(* global variable list RobotLibraryParameter *)
{attribute 'qualified_only'}
// ------------------------------------------------------------------------- 
//  SRCI Robot Library                                                
// ------------------------------------------------------------------------- 
//                                                                           
//  Object:      Parameter                                       
//  Author:      Thorsten Brach                                                
//  Date:        2024-06-01
//
//  Description:                                              
//   
//                                                                           
//  Copyright: 
//    (C) 2024 Thorsten Brach. All rights reserved                                                                                                                                            
//             Licensed under the MIT License.
//                                                                           
//  Disclaimer:                                                                           
//    This project is provided without any guarantee and can be used for   
//    private and commercial purposes. Any use is at the user’s 
//    own risk and responsibility.
//
// -------------------------------------------------------------------------
VAR_GLOBAL CONSTANT
  /// Maximal amount of tools
  TOOL_MAX                            : DINT := 16;
  /// Maximal amount of frames
  FRAME_MAX                           : DINT := 16;
  /// Maximal amount of loads
  LOAD_MAX                            : DINT := 16;  
  /// Maximal amount of work areas
  WORK_AREAS_MAX                      : DINT := 16;  
  /// Maximal amount of system logs
  SYSTEM_LOG_MAX                      : DINT := 32;  
  /// Maximal amount of message logs
  MESSAGE_LOG_MAX                     : DINT := 100;  
  /// Maximum string length for message texts
  MESSAGE_TEXT_LEN                    : DINT := 255;
  /// Maximal amount of List entries 
  LIST_ENTRIES_MAX                    : DINT := 100;
  /// Maximal amount of bytes for the parameter payload
  PARAMETER_PAYLOAD_MAX               : DINT := 255;  
  /// Maximal amount of bytes for the response payload
  RESPONSE_PAYLOAD_MAX                : DINT := 255;  
  /// Maximal amount of bytes that can be exchanged with the sub program on the RC
  SUB_PROGRAM_DATA_MAX                : DINT := 189;
  /// Maximal amount of spline data
  SPLINE_DATA_MAX                     : DINT := 64;
  /// Maximal amount of entries in the Active Command Register
  ACTIVE_CMD_REGISTER_ENTRIES_MAX     : DINT := 50;
  /// Maximal amount of message codes
  MESSAGE_CODES_MAX                   : DINT := 15;
  /// Maximal amount of fragments
  FRAGMENT_MAX                        : DINT := 9;
  /// Flag to indicate that the byte order must be changed
  SWAP_BYTE_ORDER                     : BOOL := TRUE; 
  /// Timeout for checking for invalid frames
  INVALID_FRAMES_CHECK_TIMEOUT        : TIME := T#60S;
  /// Warning limit for ACR registers running low
  ACR_USAGE_WARNING_LIMIT             : REAL := 80.0;  
END_VAR

INTERFACE IMessageLogger
METHOD PUBLIC AddMessageLog
VAR_INPUT
  /// Message to add to the log
  MessageLog : AlarmMessage;
END_VAR
END_METHOD
METHOD PUBLIC AddSystemLog
VAR_INPUT
  /// System messafe to add to the log
  SystemLog : STRING(RobotLibraryParameter.MESSAGE_TEXT_LEN);
END_VAR
END_METHOD
END_INTERFACE

INTERFACE IRobotLibraryCommandFB
METHOD PUBLIC CallBack : DINT
VAR_INPUT
  /// Response data
  RspData : AxesGroupAcyclicAcrEntryRspBuffer;  
END_VAR
END_METHOD
PROPERTY CommandData : RobotLibrarySendDataFB
END_PROPERTY
END_INTERFACE

FUNCTION IsDefaultDynamicsEqual : BOOL
// ------------------------------------------------------------------------- 
//  SRCI Robot Library                                                
// ------------------------------------------------------------------------- 
//                                                                           
//  Object:      IsDefaultDynamicsEqual                                       
//  Author:      Thorsten Brach                                                
//  Date:        2025-04-23
//
//  Description:                                              
//   
//                                                                           
//  Copyright: 
//    (C) 2025 Thorsten Brach. All rights reserved                                                                                                                                            
//             Licensed under the MIT License.
//                                                                           
//  Disclaimer:                                                                           
//    This project is provided without any guarantee and can be used for   
//    private and commercial purposes. Any use is at the user’s 
//    own risk and responsibility.
//
// -------------------------------------------------------------------------
VAR_INPUT
  /// DefaultDynamics 1 to compare
  Data1           : DefaultDynamics;
  /// DefaultDynamics 2 to compare
  Data2           : DefaultDynamics;
  /// Flag to ignore the timestamp during the comparison
  IgnoreTimestamp : BOOL;
END_VAR

            IF (IgnoreTimestamp)
THEN
  Data1.Timestamp := Data2.Timestamp;
END_IF                    
                    
IsDefaultDynamicsEqual := ( SysDepMemCmp( pData1 := ADR(Data1), pData2 :=  ADR(Data2), DataLen := SIZEOF(Data1)) = RobotLibraryConstants.OK );
          
END_FUNCTION

FUNCTION IsFrameDataEqual : BOOL
// ------------------------------------------------------------------------- 
//  SRCI Robot Library                                                
// ------------------------------------------------------------------------- 
//                                                                           
//  Object:      IsFrameDataEqual                                       
//  Author:      Thorsten Brach                                                
//  Date:        2025-04-23
//
//  Description:                                              
//   
//                                                                           
//  Copyright: 
//    (C) 2025 Thorsten Brach. All rights reserved                                                                                                                                            
//             Licensed under the MIT License.
//                                                                           
//  Disclaimer:                                                                           
//    This project is provided without any guarantee and can be used for   
//    private and commercial purposes. Any use is at the user’s 
//    own risk and responsibility.
//
// -------------------------------------------------------------------------
VAR_INPUT
  /// FrameData 1 to compare
  Data1           : FrameData;
  /// FrameData 2 to compare
  Data2           : FrameData;
  /// Flag to ignore the timestamp during the comparison
  IgnoreTimestamp : BOOL;
END_VAR

            IF (IgnoreTimestamp)
THEN
  Data1.Timestamp := Data2.Timestamp;
END_IF                    
                    
IsFrameDataEqual := ( SysDepMemCmp( pData1 := ADR(Data1), pData2 :=  ADR(Data2), DataLen := SIZEOF(Data1)) = RobotLibraryConstants.OK );                    
          
END_FUNCTION

FUNCTION IsLoadDataEqual : BOOL
// ------------------------------------------------------------------------- 
//  SRCI Robot Library                                                
// ------------------------------------------------------------------------- 
//                                                                           
//  Object:      IsLoadDataEqual                                       
//  Author:      Thorsten Brach                                                
//  Date:        2025-04-23
//
//  Description:                                              
//   
//                                                                           
//  Copyright: 
//    (C) 2025 Thorsten Brach. All rights reserved                                                                                                                                            
//             Licensed under the MIT License.
//                                                                           
//  Disclaimer:                                                                           
//    This project is provided without any guarantee and can be used for   
//    private and commercial purposes. Any use is at the user’s 
//    own risk and responsibility.
//
// -------------------------------------------------------------------------
VAR_INPUT
  /// LoadData 1 to compare
  Data1           : LoadData;
  /// LoadData 2 to compare
  Data2           : LoadData;
  /// Flag to ignore the timestamp during the comparison
  IgnoreTimestamp : BOOL;
END_VAR

            IF (IgnoreTimestamp)
THEN
  Data1.Timestamp := Data2.Timestamp;
END_IF                    
                    
IsLoadDataEqual := ( SysDepMemCmp( pData1 := ADR(Data1), pData2 :=  ADR(Data2), DataLen := SIZEOF(Data1)) = RobotLibraryConstants.OK );
          
END_FUNCTION

FUNCTION IsReferenceDynamicsEqual : BOOL
// ------------------------------------------------------------------------- 
//  SRCI Robot Library                                                
// ------------------------------------------------------------------------- 
//                                                                           
//  Object:      IsReferenceDynamicsEqual                                       
//  Author:      Thorsten Brach                                                
//  Date:        2025-04-23
//
//  Description:                                              
//   
//                                                                           
//  Copyright: 
//    (C) 2025 Thorsten Brach. All rights reserved                                                                                                                                            
//             Licensed under the MIT License.
//                                                                           
//  Disclaimer:                                                                           
//    This project is provided without any guarantee and can be used for   
//    private and commercial purposes. Any use is at the user’s 
//    own risk and responsibility.
//
// -------------------------------------------------------------------------
VAR_INPUT
  /// ReferenceDynamics 1 to compare
  Data1           : ReferenceDynamics;
  /// ReferenceDynamics 2 to compare
  Data2           : ReferenceDynamics;
  /// Flag to ignore the timestamp during the comparison
  IgnoreTimestamp : BOOL;
END_VAR

            IF (IgnoreTimestamp)
THEN
  Data1.Timestamp := Data2.Timestamp;
END_IF                    
                    
IsReferenceDynamicsEqual := ( SysDepMemCmp( pData1 := ADR(Data1), pData2 :=  ADR(Data2), DataLen := SIZEOF(Data1)) = RobotLibraryConstants.OK );
          
END_FUNCTION

FUNCTION IsSwLimitsEqual : BOOL
// ------------------------------------------------------------------------- 
//  SRCI Robot Library                                                
// ------------------------------------------------------------------------- 
//                                                                           
//  Object:      IsSwLimitsEqual                                       
//  Author:      Thorsten Brach                                                
//  Date:        2025-04-23
//
//  Description:                                              
//   
//                                                                           
//  Copyright: 
//    (C) 2025 Thorsten Brach. All rights reserved                                                                                                                                            
//             Licensed under the MIT License.
//                                                                           
//  Disclaimer:                                                                           
//    This project is provided without any guarantee and can be used for   
//    private and commercial purposes. Any use is at the user’s 
//    own risk and responsibility.
//
// -------------------------------------------------------------------------
VAR_INPUT
  /// SW Limit 1 to compare
  Data1           : SWLimits;
  /// SW LIMIT 2 to compare
  Data2           : SWLimits;
  /// Flag to ignore the timestamp during the comparison
  IgnoreTimestamp : BOOL;
END_VAR

            IF (IgnoreTimestamp)
THEN
  Data1.Timestamp := Data2.Timestamp;
END_IF                    
                    
IsSwLimitsEqual := ( SysDepMemCmp( pData1 := ADR(Data1), pData2 :=  ADR(Data2), DataLen := SIZEOF(Data1)) = RobotLibraryConstants.OK );
          
END_FUNCTION

FUNCTION IsToolDataEqual : BOOL
// ------------------------------------------------------------------------- 
//  SRCI Robot Library                                                
// ------------------------------------------------------------------------- 
//                                                                           
//  Object:      IsToolDataEqual                                       
//  Author:      Thorsten Brach                                                
//  Date:        2025-04-23
//
//  Description:                                              
//   
//                                                                           
//  Copyright: 
//    (C) 2025 Thorsten Brach. All rights reserved                                                                                                                                            
//             Licensed under the MIT License.
//                                                                           
//  Disclaimer:                                                                           
//    This project is provided without any guarantee and can be used for   
//    private and commercial purposes. Any use is at the user’s 
//    own risk and responsibility.
//
// -------------------------------------------------------------------------
VAR_INPUT
  /// ToolData 1 to compare
  Data1           : ToolData;
  /// ToolData 2 to compare
  Data2           : ToolData;
  /// Flag to ignore the timestamp during the comparison
  IgnoreTimestamp : BOOL;
END_VAR

            IF (IgnoreTimestamp)
THEN
  Data1.Timestamp := Data2.Timestamp;
END_IF                    
                    
IsToolDataEqual := ( SysDepMemCmp( pData1 := ADR(Data1), pData2 :=  ADR(Data2), DataLen := SIZEOF(Data1)) = RobotLibraryConstants.OK );                    
          
END_FUNCTION

FUNCTION IsWorkAreaEqual : BOOL
// ------------------------------------------------------------------------- 
//  SRCI Robot Library                                                
// ------------------------------------------------------------------------- 
//                                                                           
//  Object:      IsWorkAreaEqual                                       
//  Author:      Thorsten Brach                                                
//  Date:        2025-04-23
//
//  Description:                                              
//   
//                                                                           
//  Copyright: 
//    (C) 2025 Thorsten Brach. All rights reserved                                                                                                                                            
//             Licensed under the MIT License.
//                                                                           
//  Disclaimer:                                                                           
//    This project is provided without any guarantee and can be used for   
//    private and commercial purposes. Any use is at the user’s 
//    own risk and responsibility.
//
// -------------------------------------------------------------------------
VAR_INPUT
  /// WorkArea 1 to compare
  Data1           : RobotWorkAreaData;
  /// WorkArea 2 to compare
  Data2           : RobotWorkAreaData;
  /// Flag to ignore the timestamp during the comparison
  IgnoreTimestamp : BOOL;
END_VAR

            IF (IgnoreTimestamp)
THEN
  Data1.Timestamp := Data2.Timestamp;
END_IF                    
                    
IsWorkAreaEqual := ( SysDepMemCmp( pData1 := ADR(Data1), pData2 :=  ADR(Data2), DataLen := SIZEOF(Data1)) = RobotLibraryConstants.OK );
          
END_FUNCTION

FUNCTION CheckTimeout : DINT
// ------------------------------------------------------------------------- 
//  SRCI Robot Library                                                
// ------------------------------------------------------------------------- 
//                                                                           
//  Object:      SwapBytes                                       
//  Author:      Thorsten Brach                                                
//  Date:        2024-12-18
//
//  Description:                                              
//   
//                                                                           
//  Copyright: 
//    (C) 2024 Thorsten Brach. All rights reserved                                                                                                                                            
//             Licensed under the MIT License.
//                                                                           
//  Disclaimer:                                                                           
//    This project is provided without any guarantee and can be used for   
//    private and commercial purposes. Any use is at the user’s 
//    own risk and responsibility.
//
// -------------------------------------------------------------------------
VAR_INPUT
  /// Reference to TON instance
  rTimer : REFERENCE TO TON;
END_VAR

            // Call timer 
rTimer();

// check if timer elapsed
IF (rTimer.Q = TRUE)
THEN
  // assign return value
  CheckTimeout := RobotLibraryConstants.OK;
ELSE
  // assign return value
  CheckTimeout := RobotLibraryConstants.RUNNING;
END_IF
          
END_FUNCTION

FUNCTION SetTimeout : DINT
// ------------------------------------------------------------------------- 
//  SRCI Robot Library                                                
// ------------------------------------------------------------------------- 
//                                                                           
//  Object:      SwapBytes                                       
//  Author:      Thorsten Brach                                                
//  Date:        2024-12-18
//
//  Description:                                              
//   
//                                                                           
//  Copyright: 
//    (C) 2024 Thorsten Brach. All rights reserved                                                                                                                                            
//             Licensed under the MIT License.
//                                                                           
//  Disclaimer:                                                                           
//    This project is provided without any guarantee and can be used for   
//    private and commercial purposes. Any use is at the user’s 
//    own risk and responsibility.
//
// -------------------------------------------------------------------------
VAR_INPUT
  /// Timeout to be set
  PT     : TIME;
  /// Reference to TON instance
  rTimer : REFERENCE TO TON;
END_VAR

            rTimer(IN := FALSE);          // Reset timer
rTimer(PT := PT, IN := TRUE); // Start timer

// assign return value
SetTimeout := RobotLibraryConstants.OK;
          
END_FUNCTION

FUNCTION DATE_TO_IEC_DATE : IEC_DATE
// ------------------------------------------------------------------------- 
//  SRCI Robot Library                                                
// ------------------------------------------------------------------------- 
//                                                                           
//  Object:      DATE_TO_IEC_DATE                                       
//  Author:      Thorsten Brach                                                
//  Date:        2024-06-01
//
//  Description:                                              
//   
//                                                                           
//  Copyright: 
//    (C) 2024 Thorsten Brach. All rights reserved                                                                                                                                            
//             Licensed under the MIT License.
//                                                                           
//  Disclaimer:                                                                           
//    This project is provided without any guarantee and can be used for   
//    private and commercial purposes. Any use is at the user’s 
//    own risk and responsibility.
//
// -------------------------------------------------------------------------
VAR_INPUT
  Value    : DATE;
END_VAR

VAR
 _tmpDate1 : DWORD;
 _tmpDate2 : DWORD;
 _initDate : DATE := DATE#1990-01-01;
 END_VAR

            // Siemens Dateformat is Day since 01.01.1990
// TwinCat Dateformat is seconds sinde 01.01.1970
// Calculation : 
// ( [TwinCat current date] - [ TwinCat 01.01.1970] ) / [Seconds a Day] = Days sinde 01.01.1990 (Siemens Format)

// copy date to dword
SysDepMemCpy( pDest := ADR(_tmpDate1), pSrc := ADR( Value   ), DataLen := SIZEOF( Value   ));
// copy date to dword
SysDepMemCpy( pDest := ADR(_tmpDate2), pSrc := ADR(_initDate), DataLen := SIZEOF(_initDate));

// calculate IEC Date :  
DATE_TO_IEC_DATE := UDINT_TO_UINT((_tmpDate1 - _tmpDate2) / 86400); // 86400 Seconds = 1 day 

          
END_FUNCTION

FUNCTION IEC_DATE_TO_DATE : DATE
// ------------------------------------------------------------------------- 
//  SRCI Robot Library                                                
// ------------------------------------------------------------------------- 
//                                                                           
//  Object:      IEC_DATE_TO_DATE                                       
//  Author:      Thorsten Brach                                                
//  Date:        2025-01-05
//
//  Description:                                              
//   
//                                                                           
//  Copyright: 
//    (C) 2025 Thorsten Brach. All rights reserved                                                                                                                                            
//             Licensed under the MIT License.
//                                                                           
//  Disclaimer:                                                                           
//    This project is provided without any guarantee and can be used for   
//    private and commercial purposes. Any use is at the user’s 
//    own risk and responsibility.
//
// -------------------------------------------------------------------------
VAR_INPUT
  Value    : IEC_DATE;
END_VAR

VAR
 _tmpDate1 : DWORD;
 _initDate : DATE := DATE#1990-01-01;
 END_VAR

            // Siemens Dateformat is Day since 01.01.1990
// TwinCat Dateformat is seconds sinde 01.01.1970
// Calculation : 
// ( [ TwinCat 01.01.1990] + [IEC Date]) * [Seconds a Day] = (TwinCat Format)

// copy date to dword
SysDepMemCpy( pDest := ADR(_tmpDate1), pSrc := ADR( _initDate ), DataLen := SIZEOF( _initDate ));

// calculate IEC Date :  
IEC_DATE_TO_DATE := DWORD_TO_DATE( _tmpDate1 + ( Value * 86400)); // 86400 Seconds = 1 day 
          
END_FUNCTION

FUNCTION IEC_TIME_TO_TIME : TOD
// ------------------------------------------------------------------------- 
//  SRCI Robot Library                                                
// ------------------------------------------------------------------------- 
//                                                                           
//  Object:      IEC_TIME_TO_TIME                                       
//  Author:      Thorsten Brach                                                
//  Date:        2025-01-05
//
//  Description:                                              
//   
//                                                                           
//  Copyright: 
//    (C) 2025 Thorsten Brach. All rights reserved                                                                                                                                            
//             Licensed under the MIT License.
//                                                                           
//  Disclaimer:                                                                           
//    This project is provided without any guarantee and can be used for   
//    private and commercial purposes. Any use is at the user’s 
//    own risk and responsibility.
//
// -------------------------------------------------------------------------
VAR_INPUT
  Value : IEC_TIME;
END_VAR

            IEC_TIME_TO_TIME := Value; 
          
END_FUNCTION

FUNCTION IEC_TIMESTAMP_TO_DT : DT
// ------------------------------------------------------------------------- 
//  SRCI Robot Library                                                
// ------------------------------------------------------------------------- 
//                                                                           
//  Object:      TIME_TO_IEC_TIME                                       
//  Author:      Thorsten Brach                                                
//  Date:        2025-01-05
//
//  Description:                                              
//   
//                                                                           
//  Copyright: 
//    (C) 2025 Thorsten Brach. All rights reserved                                                                                                                                            
//             Licensed under the MIT License.
//                                                                           
//  Disclaimer:                                                                           
//    This project is provided without any guarantee and can be used for   
//    private and commercial purposes. Any use is at the user’s 
//    own risk and responsibility.
//
// -------------------------------------------------------------------------
VAR_INPUT
  Value : IEC_TIMESTAMP;
END_VAR

VAR
  /// internal date
 _date    : DATE;
  /// internal date as string
 _dateStr : STRING;
  /// internal time
 _time    : TOD;
  /// internal time as string
 _timeStr : STRING;
END_VAR

            _date := IEC_DATE_TO_DATE(Value.IEC_DATE); 
_time := IEC_TIME_TO_TIME(Value.IEC_TIME); 


// Example : DATE#2025-1-5
_dateStr := DATE_TO_STRING(_date);
// Example : DT#2025-1-5
_dateStr := strReplace(_dateStr, 'D#', 'DT#');

// Example : TOD#15:18:4.567
_timeStr :=  TOD_TO_STRING(_time);
// Example : -15:18:4.567
_timeStr := strReplace(_timeStr, 'TOD#', '-');

// Example : DT#2025-1-5-15:18:4.567
IEC_TIMESTAMP_TO_DT := STRING_TO_DT( Concat(_dateStr,_timeStr));
          
END_FUNCTION

FUNCTION IEC_TIMESTAMP_TO_SYSTEMTIME : SystemTime
// ------------------------------------------------------------------------- 
//  SRCI Robot Library                                                
// ------------------------------------------------------------------------- 
//                                                                           
//  Object:      IEC_TIMESTAMP_TO_SYSTEMTIME                                       
//  Author:      Thorsten Brach                                                
//  Date:        2025-01-05
//
//  Description:                                              
//   
//                                                                           
//  Copyright: 
//    (C) 2025 Thorsten Brach. All rights reserved                                                                                                                                            
//             Licensed under the MIT License.
//                                                                           
//  Disclaimer:                                                                           
//    This project is provided without any guarantee and can be used for   
//    private and commercial purposes. Any use is at the user’s 
//    own risk and responsibility.
//
// -------------------------------------------------------------------------
VAR_INPUT
  Value : IEC_TIMESTAMP;
END_VAR

VAR
  /// internal date
 _date    : DATE;
  /// internal date as string
 _dateStr : STRING;
  /// internal time
 _time    : TOD;
  /// internal time as string
 _timeStr : STRING;
END_VAR

            IEC_TIMESTAMP_TO_SYSTEMTIME.SystemDate := IEC_DATE_TO_DATE(Value.IEC_DATE);
IEC_TIMESTAMP_TO_SYSTEMTIME.SystemTime := IEC_TIME_TO_TIME(Value.IEC_TIME);
          
END_FUNCTION

FUNCTION SYSTEMTIME_TO_IEC_TIMESTAMP : IEC_TIMESTAMP
// ------------------------------------------------------------------------- 
//  SRCI Robot Library                                                
// ------------------------------------------------------------------------- 
//                                                                           
//  Object:      SYSTEMTIME_TO_IEC_TIMESTAMP                                       
//  Author:      Thorsten Brach                                                
//  Date:        2025-03-30
//
//  Description:                                              
//   
//                                                                           
//  Copyright: 
//    (C) 2025 Thorsten Brach. All rights reserved                                                                                                                                            
//             Licensed under the MIT License.
//                                                                           
//  Disclaimer:                                                                           
//    This project is provided without any guarantee and can be used for   
//    private and commercial purposes. Any use is at the user’s 
//    own risk and responsibility.
//
// -------------------------------------------------------------------------
VAR_INPUT
  SystemTime : SystemTime;
END_VAR

            SYSTEMTIME_TO_IEC_TIMESTAMP.IEC_DATE := DATE_TO_IEC_DATE(SystemTime.SystemDate);
SYSTEMTIME_TO_IEC_TIMESTAMP.IEC_TIME := TIME_TO_IEC_TIME(SystemTime.SystemTime);

          
END_FUNCTION

FUNCTION TIME_TO_IEC_TIME : IEC_TIME
// ------------------------------------------------------------------------- 
//  SRCI Robot Library                                                
// ------------------------------------------------------------------------- 
//                                                                           
//  Object:      TIME_TO_IEC_TIME                                       
//  Author:      Thorsten Brach                                                
//  Date:        2024-06-01
//
//  Description:                                              
//   
//                                                                           
//  Copyright: 
//    (C) 2024 Thorsten Brach. All rights reserved                                                                                                                                            
//             Licensed under the MIT License.
//                                                                           
//  Disclaimer:                                                                           
//    This project is provided without any guarantee and can be used for   
//    private and commercial purposes. Any use is at the user’s 
//    own risk and responsibility.
//
// -------------------------------------------------------------------------
VAR_INPUT
  Value : TOD;
END_VAR

            TIME_TO_IEC_TIME := Value; 
          
END_FUNCTION

FUNCTION ArmConfigParameterToBytes : ARRAY[0..1] of BYTE
// ------------------------------------------------------------------------- 
//  SRCI Robot Library                                                
// ------------------------------------------------------------------------- 
//                                                                           
//  Object:      ArmConfigParameterToBytes                                       
//  Author:      Thorsten Brach                                                
//  Date:        2025-01-30
//
//  Description:                                              
//   
//                                                                           
//  Copyright: 
//    (C) 2025 Thorsten Brach. All rights reserved                                                                                                                                            
//             Licensed under the MIT License.
//                                                                           
//  Disclaimer:                                                                           
//    This project is provided without any guarantee and can be used for   
//    private and commercial purposes. Any use is at the user’s 
//    own risk and responsibility.
//
// -------------------------------------------------------------------------
VAR_INPUT
 /// ArmConfigParameter
 Value: ArmConfigParameter;
END_VAR

            ArmConfigParameterToBytes[0].0 := Value.Shoulder.0;
ArmConfigParameterToBytes[0].1 := Value.Shoulder.1;
ArmConfigParameterToBytes[0].2 := Value.Shoulder.2;
ArmConfigParameterToBytes[0].3 := Value.Shoulder.3;
ArmConfigParameterToBytes[0].4 := Value.Elbow.0;
ArmConfigParameterToBytes[0].5 := Value.Elbow.1;
ArmConfigParameterToBytes[0].6 := Value.Elbow.2;
ArmConfigParameterToBytes[0].7 := Value.Elbow.3;
ArmConfigParameterToBytes[1].0 := Value.Wrist.0;
ArmConfigParameterToBytes[1].1 := Value.Wrist.1;
ArmConfigParameterToBytes[1].2 := Value.Wrist.2;
ArmConfigParameterToBytes[1].3 := Value.Wrist.3;
ArmConfigParameterToBytes[1].4 := FALSE;
ArmConfigParameterToBytes[1].5 := FALSE;
ArmConfigParameterToBytes[1].6 := FALSE;
ArmConfigParameterToBytes[1].7 := FALSE;
          
END_FUNCTION

FUNCTION BytesToRCSupportedFunctions : RCSupportedFunctions
// ------------------------------------------------------------------------- 
//  SRCI Robot Library                                                
// ------------------------------------------------------------------------- 
//                                                                           
//  Object:      BytesToRCSupportedFunctions                                       
//  Author:      Thorsten Brach                                                
//  Date:        2024-12-18
//
//  Description:                                              
//   
//                                                                           
//  Copyright: 
//    (C) 2024 Thorsten Brach. All rights reserved                                                                                                                                            
//             Licensed under the MIT License.
//                                                                           
//  Disclaimer:                                                                           
//    This project is provided without any guarantee and can be used for   
//    private and commercial purposes. Any use is at the user’s 
//    own risk and responsibility.
//
// -------------------------------------------------------------------------
VAR_INPUT
  Bytes : ARRAY [0..18] OF BYTE;
END_VAR

            // Byte 00 - Bit 0  
BytesToRCSupportedFunctions.Reserved                   := Bytes[00].0;
// Byte 00 - Bit 1 
BytesToRCSupportedFunctions.ReadRobotData              := Bytes[00].1;
// Byte 00 - Bit 2  
BytesToRCSupportedFunctions.EnableRobot                := Bytes[00].2;
// Byte 00 - Bit 3  
BytesToRCSupportedFunctions.GroupReset                 := Bytes[00].3;
// Byte 00 - Bit 4  
BytesToRCSupportedFunctions.ReadActualPosition         := Bytes[00].4;
// Byte 00 - Bit 5 
BytesToRCSupportedFunctions.ReadActualPositionCyclic   := Bytes[00].5;
// Byte 00 - Bit 6  
BytesToRCSupportedFunctions.ExchangeConfiguration      := Bytes[00].6;
// Byte 00 - Bit 7  
BytesToRCSupportedFunctions.SetSequence                := Bytes[00].7;

// Byte 01 - Bit 0  
BytesToRCSupportedFunctions.ChangeSpeedOverride        := Bytes[01].0;
// Byte 01 - Bit 1  
BytesToRCSupportedFunctions.ReadMessages               := Bytes[01].1;
// Byte 01 - Bit 2  
BytesToRCSupportedFunctions.ReadRobotReferenceDynamics := Bytes[01].2;
// Byte 01 - Bit 3  
BytesToRCSupportedFunctions.WriteFrameData             := Bytes[01].3;
// Byte 01 - Bit 4  
BytesToRCSupportedFunctions.WriteToolData              := Bytes[01].4;
// Byte 01 - Bit 5  
BytesToRCSupportedFunctions.WriteLoadData              := Bytes[01].5;
// Byte 01 - Bit 6  
BytesToRCSupportedFunctions.WriteRobotReferenceDynamics:= Bytes[01].6;
// Byte 01 - Bit 7  
BytesToRCSupportedFunctions.WriteRobotDefaultDynamics  := Bytes[01].7;

// Byte 02 - Bit 0  
BytesToRCSupportedFunctions.ReadRobotDefaultDynamics   := Bytes[02].0;
// Byte 02 - Bit 1  
BytesToRCSupportedFunctions.ReadFrameData              := Bytes[02].1;
// Byte 02 - Bit 2  
BytesToRCSupportedFunctions.ReadToolData               := Bytes[02].2;
// Byte 02 - Bit 3  
BytesToRCSupportedFunctions.ReadLoadData               := Bytes[02].3;
// Byte 02 - Bit 4  
BytesToRCSupportedFunctions.ReadRobotSWLimits          := Bytes[02].4;
// Byte 02 - Bit 5  
BytesToRCSupportedFunctions.GroupJog                   := Bytes[02].5;
// Byte 02 - Bit 6  
BytesToRCSupportedFunctions.MoveLinearAbsolute         := Bytes[02].6;
// Byte 02 - Bit 7  
BytesToRCSupportedFunctions.MoveDirectAbsolute         := Bytes[02].7;

// Byte 03 - Bit 0  
BytesToRCSupportedFunctions.MoveAxesAbsolute           := Bytes[03].0;
// Byte 03 - Bit 1  
BytesToRCSupportedFunctions.GroupStop                  := Bytes[03].1;
// Byte 03 - Bit 2
BytesToRCSupportedFunctions.GroupContinue              := Bytes[03].2;
// Byte 03 - Bit 3
BytesToRCSupportedFunctions.GroupInterrupt             := Bytes[03].3;
// Byte 03 - Bit 4
BytesToRCSupportedFunctions.ReturnToPrimary            := Bytes[03].4;
// Byte 03 - Bit 5
BytesToRCSupportedFunctions.MoveLinearAbsoluteJ        := Bytes[03].5;
// Byte 03 - Bit 6
BytesToRCSupportedFunctions.MoveDirectRelative         := Bytes[03].6;
// Byte 03 - Bit 7
BytesToRCSupportedFunctions.MoveAxesRelative           := Bytes[03].7;

// Byte 04 - Bit 0
BytesToRCSupportedFunctions.MoveCircularAbsolute       := Bytes[04].0;
// Byte 04 - Bit 1
BytesToRCSupportedFunctions.MoveCircularRelative       := Bytes[04].1;
// Byte 04 - Bit 2
BytesToRCSupportedFunctions.MoveLinearOffset           := Bytes[04].2;
// Byte 04 - Bit 3
BytesToRCSupportedFunctions.MoveDirectOffset           := Bytes[04].3;
// Byte 04 - Bit 4
BytesToRCSupportedFunctions.WaitTime                   := Bytes[04].4;
// Byte 04 - Bit 5
BytesToRCSupportedFunctions.ReadDigitalInputs          := Bytes[04].5;
// Byte 04 - Bit 6
BytesToRCSupportedFunctions.ReadDigitalOutputs         := Bytes[04].6;
// Byte 04 - Bit 7
BytesToRCSupportedFunctions.WriteDigitalOutputs        := Bytes[04].7;

// Byte 05 - Bit 0
BytesToRCSupportedFunctions.ReadIntegers               := Bytes[05].0;
// Byte 05 - Bit 1
BytesToRCSupportedFunctions.ReadReals                  := Bytes[05].1;
// Byte 05 - Bit 2
BytesToRCSupportedFunctions.WriteIntegers              := Bytes[05].2;
// Byte 05 - Bit 3
BytesToRCSupportedFunctions.WriteReals                 := Bytes[05].3;
// Byte 05 - Bit 4
BytesToRCSupportedFunctions.MoveLinearCam              := Bytes[05].4;
// Byte 05 - Bit 5
BytesToRCSupportedFunctions.MoveDirectCam              := Bytes[05].5;
// Byte 05 - Bit 6
BytesToRCSupportedFunctions.MoveCircularCam            := Bytes[05].6;
// Byte 05 - Bit 7
BytesToRCSupportedFunctions.SetTriggerRegister         := Bytes[05].7;

// Byte 06 - Bit 0
BytesToRCSupportedFunctions.SetTriggerLimit            := Bytes[06].0;
// Byte 06 - Bit 1
BytesToRCSupportedFunctions.SetTriggerUser             := Bytes[06].1;
// Byte 06 - Bit 2
BytesToRCSupportedFunctions.SetTriggerError            := Bytes[06].2;
// Byte 06 - Bit 3
BytesToRCSupportedFunctions.ReactAtTrigger             := Bytes[06].3;
// Byte 06 - Bit 4
BytesToRCSupportedFunctions.WaitForTrigger             := Bytes[06].4;
// Byte 06 - Bit 5
BytesToRCSupportedFunctions.ReadSystemVariable         := Bytes[06].5;
// Byte 06 - Bit 6
BytesToRCSupportedFunctions.WriteSystemVariable        := Bytes[06].6;
// Byte 06 - Bit 7
BytesToRCSupportedFunctions.CalculateForwardKinematic  := Bytes[06].7;

// Byte 07 - Bit 0
BytesToRCSupportedFunctions.CalculateInverseKinematic  := Bytes[07].0;
// Byte 07 - Bit 1
BytesToRCSupportedFunctions.CalculateCartesianPosition := Bytes[07].1;
// Byte 07 - Bit 2
BytesToRCSupportedFunctions.CalculateTool              := Bytes[07].2;
// Byte 07 - Bit 3
BytesToRCSupportedFunctions.CalculateFrame             := Bytes[07].3;
// Byte 07 - Bit 4
BytesToRCSupportedFunctions.ActivateNextCommand        := Bytes[07].4;
// Byte 07 - Bit 5
BytesToRCSupportedFunctions.ShiftPosition              := Bytes[07].5;
// Byte 07 - Bit 6
BytesToRCSupportedFunctions.CallSubprogram             := Bytes[07].6;
// Byte 07 - Bit 7
BytesToRCSupportedFunctions.MoveLinearRelative         := Bytes[07].7;

// Byte 08 - Bit 0
BytesToRCSupportedFunctions.WriteCallSubprogramCyclic  := Bytes[08].0;
// Byte 08 - Bit 1
BytesToRCSupportedFunctions.ReadCallSubprogramCyclic   := Bytes[08].1;
// Byte 08 - Bit 2
BytesToRCSupportedFunctions.StopSubprogram             := Bytes[08].2;
// Byte 08 - Bit 3
BytesToRCSupportedFunctions.ReadDHParameter            := Bytes[08].3;
// Byte 08 - Bit 4
BytesToRCSupportedFunctions.RestartController          := Bytes[08].4;
// Byte 08 - Bit 5
BytesToRCSupportedFunctions.ReadActualTCPVelocity      := Bytes[08].5;
// Byte 08 - Bit 6
BytesToRCSupportedFunctions.UserLogin                  := Bytes[08].6;
// Byte 08 - Bit 7
BytesToRCSupportedFunctions.SwitchLanguage             := Bytes[08].7;

// Byte 09 - Bit 0
BytesToRCSupportedFunctions.WriteRobotSWLimits         := Bytes[09].0;
// Byte 09 - Bit 1
BytesToRCSupportedFunctions.SetOperationMode           := Bytes[09].1;
// Byte 09 - Bit 2
BytesToRCSupportedFunctions.ReadWorkArea               := Bytes[09].2;
// Byte 09 - Bit 3
BytesToRCSupportedFunctions.WriteWorkArea              := Bytes[09].3;
// Byte 09 - Bit 4
BytesToRCSupportedFunctions.ActivateWorkArea           := Bytes[09].4;
// Byte 09 - Bit 5
BytesToRCSupportedFunctions.MonitorWorkArea            := Bytes[09].5;
// Byte 09 - Bit 6
BytesToRCSupportedFunctions.MoveApproachLinear         := Bytes[09].6;
// Byte 09 - Bit 7
BytesToRCSupportedFunctions.MoveDepartLinear           := Bytes[09].7;

// Byte 10 - Bit 0
BytesToRCSupportedFunctions.MoveApproachDirect         := Bytes[10].0;
// Byte 10 - Bit 1
BytesToRCSupportedFunctions.MoveDepartDirect           := Bytes[10].1;
// Byte 10 - Bit 2
BytesToRCSupportedFunctions.SearchHardstop             := Bytes[10].2;
// Byte 10 - Bit 3
BytesToRCSupportedFunctions.SearchHardstopJ            := Bytes[10].3;
// Byte 10 - Bit 4
BytesToRCSupportedFunctions.MovePickPlaceLinear        := Bytes[10].4;
// Byte 10 - Bit 5
BytesToRCSupportedFunctions.MovePickPlaceDirect        := Bytes[10].5;
// Byte 10 - Bit 6
BytesToRCSupportedFunctions.ActivateConveyorTracking   := Bytes[10].6;
// Byte 10 - Bit 7
BytesToRCSupportedFunctions.RedefineTrackingPosition   := Bytes[10].7;

// Byte 11 - Bit 0
BytesToRCSupportedFunctions.SyncToConveyor             := Bytes[11].0;
// Byte 11 - Bit 1
BytesToRCSupportedFunctions.ConfigureConveyor          := Bytes[11].1;
// Byte 11 - Bit 2
BytesToRCSupportedFunctions.MoveSuperImposed           := Bytes[11].2;
// Byte 11 - Bit 3
BytesToRCSupportedFunctions.MoveSuperImposedDynamic    := Bytes[11].3;
// Byte 11 - Bit 4
BytesToRCSupportedFunctions.ReadAnalogInput            := Bytes[11].4;
// Byte 11 - Bit 5
BytesToRCSupportedFunctions.ReadAnalogOutput           := Bytes[11].5;
// Byte 11 - Bit 6
BytesToRCSupportedFunctions.WriteAnalogOutput          := Bytes[11].6;
// Byte 11 - Bit 7
BytesToRCSupportedFunctions.MeasuringInput             := Bytes[11].7;

// Byte 12 - Bit 0
BytesToRCSupportedFunctions.AbortMeasuringInput        := Bytes[12].0;
// Byte 12 - Bit 1
BytesToRCSupportedFunctions.SetTriggerMotion           := Bytes[12].1;
// Byte 12 - Bit 2
BytesToRCSupportedFunctions.OpenBrake                  := Bytes[12].2;
// Byte 12 - Bit 3
BytesToRCSupportedFunctions.PathAccuracyMode           := Bytes[12].3;
// Byte 12 - Bit 4
BytesToRCSupportedFunctions.AvoidSingularity           := Bytes[12].4;
// Byte 12 - Bit 5
BytesToRCSupportedFunctions.ForceControl               := Bytes[12].5;
// Byte 12 - Bit 6
BytesToRCSupportedFunctions.ForceLimit                 := Bytes[12].6;
// Byte 12 - Bit 7
BytesToRCSupportedFunctions.ReadActualForce            := Bytes[12].7;

// Byte 13 - Bit 0
BytesToRCSupportedFunctions.BrakeTest                  := Bytes[13].0;
// Byte 13 - Bit 1
BytesToRCSupportedFunctions.SoftSwitchTCP              := Bytes[13].1;
// Byte 13 - Bit 2
BytesToRCSupportedFunctions.CreateSpline               := Bytes[13].2;
// Byte 13 - Bit 3
BytesToRCSupportedFunctions.DeleteSpline               := Bytes[13].3;
// Byte 13 - Bit 4
BytesToRCSupportedFunctions.MoveSpline                 := Bytes[13].4;
// Byte 13 - Bit 5
BytesToRCSupportedFunctions.DynamicSpline              := Bytes[13].5;
// Byte 13 - Bit 6
BytesToRCSupportedFunctions.LoadMeasurementAutomatic   := Bytes[13].6;
// Byte 13 - Bit 7
BytesToRCSupportedFunctions.LoadMeasurementSequential  := Bytes[13].7;

// Byte 14 - Bit 0
BytesToRCSupportedFunctions.CollisionDetection         := Bytes[14].0;
// Byte 14 - Bit 1
BytesToRCSupportedFunctions.FreeDrive                  := Bytes[14].1;
// Byte 14 - Bit 2
BytesToRCSupportedFunctions.UnitMeasurement            := Bytes[14].2;
// Byte 14 - Bit 3
BytesToRCSupportedFunctions.Byte14Bit03                := Bytes[14].3;
// Byte 14 - Bit 4
BytesToRCSupportedFunctions.Byte14Bit04                := Bytes[14].4;
// Byte 14 - Bit 5
BytesToRCSupportedFunctions.Byte14Bit05                := Bytes[14].5;
// Byte 14 - Bit 6
BytesToRCSupportedFunctions.Byte14Bit06                := Bytes[14].6;
// Byte 14 - Bit 7
BytesToRCSupportedFunctions.Byte14Bit07                := Bytes[14].7;

// Byte 15 - Bit 0
BytesToRCSupportedFunctions.Byte15Bit00                := Bytes[15].0;
// Byte 15 - Bit 1
BytesToRCSupportedFunctions.Byte15Bit01                := Bytes[15].1;
// Byte 15 - Bit 2
BytesToRCSupportedFunctions.Byte15Bit02                := Bytes[15].2;
// Byte 15 - Bit 3
BytesToRCSupportedFunctions.Byte15Bit03                := Bytes[15].3;
// Byte 15 - Bit 4
BytesToRCSupportedFunctions.Byte15Bit04                := Bytes[15].4;
// Byte 15 - Bit 5
BytesToRCSupportedFunctions.Byte15Bit05                := Bytes[15].5;
// Byte 15 - Bit 6
BytesToRCSupportedFunctions.Byte15Bit06                := Bytes[15].6;
// Byte 15 - Bit 7
BytesToRCSupportedFunctions.Byte15Bit07                := Bytes[15].7;

// Byte 16 - Bit 0
BytesToRCSupportedFunctions.Byte16Bit00                := Bytes[16].0;
// Byte 15 - Bit 1
BytesToRCSupportedFunctions.Byte16Bit01                := Bytes[16].1;
// Byte 15 - Bit 2
BytesToRCSupportedFunctions.Byte16Bit02                := Bytes[16].2;
// Byte 15 - Bit 3
BytesToRCSupportedFunctions.Byte16Bit03                := Bytes[16].3;
// Byte 15 - Bit 4
BytesToRCSupportedFunctions.Byte16Bit04                := Bytes[16].4;
// Byte 15 - Bit 5
BytesToRCSupportedFunctions.Byte16Bit05                := Bytes[16].5;
// Byte 15 - Bit 6
BytesToRCSupportedFunctions.Byte16Bit06                := Bytes[16].6;
// Byte 15 - Bit 7
BytesToRCSupportedFunctions.Byte16Bit07                := Bytes[16].7;

// Byte 17 - Bit 0
BytesToRCSupportedFunctions.Byte17Bit00                := Bytes[17].0;
// Byte 17 - Bit 1
BytesToRCSupportedFunctions.Byte17Bit01                := Bytes[17].1;
// Byte 17 - Bit 2
BytesToRCSupportedFunctions.Byte17Bit02                := Bytes[17].2;
// Byte 17 - Bit 3
BytesToRCSupportedFunctions.Byte17Bit03                := Bytes[17].3;
// Byte 17 - Bit 4
BytesToRCSupportedFunctions.Byte17Bit04                := Bytes[17].4;
// Byte 17 - Bit 5
BytesToRCSupportedFunctions.Byte17Bit05                := Bytes[17].5;
// Byte 17 - Bit 6
BytesToRCSupportedFunctions.Byte17Bit06                := Bytes[17].6;
// Byte 17 - Bit 7
BytesToRCSupportedFunctions.Byte17Bit07                := Bytes[17].7;

// Byte 18 - Bit 0
BytesToRCSupportedFunctions.Byte18Bit00                := Bytes[18].0;
// Byte 18 - Bit 1
BytesToRCSupportedFunctions.Byte18Bit01                := Bytes[18].1;
// Byte 18 - Bit 2
BytesToRCSupportedFunctions.Byte18Bit02                := Bytes[18].2;
// Byte 18 - Bit 3
BytesToRCSupportedFunctions.Byte18Bit03                := Bytes[18].3;
// Byte 18 - Bit 4
BytesToRCSupportedFunctions.Byte18Bit04                := Bytes[18].4;
// Byte 18 - Bit 5
BytesToRCSupportedFunctions.Byte18Bit05                := Bytes[18].5;
// Byte 18 - Bit 6
BytesToRCSupportedFunctions.Byte18Bit06                := Bytes[18].6;
// Byte 18 - Bit 7
BytesToRCSupportedFunctions.Byte18Bit07                := Bytes[18].7;
          
END_FUNCTION

FUNCTION ByteToAxisExternalUnit : AxisExternalUnit
// ------------------------------------------------------------------------- 
//  SRCI Robot Library                                                
// ------------------------------------------------------------------------- 
//                                                                           
//  Object:      ByteToAxisExternalUnit                                       
//  Author:      Thorsten Brach                                                
//  Date:        2025-03-23
//
//  Description:                                              
//   
//                                                                           
//  Copyright: 
//    (C) 2025 Thorsten Brach. All rights reserved                                                                                                                                            
//             Licensed under the MIT License.
//                                                                           
//  Disclaimer:                                                                           
//    This project is provided without any guarantee and can be used for   
//    private and commercial purposes. Any use is at the user’s 
//    own risk and responsibility.
//
// -------------------------------------------------------------------------
VAR_INPUT
  AxisExternalUnit : BYTE;
END_VAR

            ByteToAxisExternalUnit.E1.0 := AxisExternalUnit.1;
ByteToAxisExternalUnit.E2.0 := AxisExternalUnit.2;
ByteToAxisExternalUnit.E3.0 := AxisExternalUnit.3;
ByteToAxisExternalUnit.E4.0 := AxisExternalUnit.4;
ByteToAxisExternalUnit.E5.0 := AxisExternalUnit.5;
ByteToAxisExternalUnit.E6.0 := AxisExternalUnit.6;
          
END_FUNCTION

FUNCTION ByteToAxisExternalUsed : AxisExternalUsed
// ------------------------------------------------------------------------- 
//  SRCI Robot Library                                                
// ------------------------------------------------------------------------- 
//                                                                           
//  Object:      ByteToAxisExternalUsed                                       
//  Author:      Thorsten Brach                                                
//  Date:        2025-03-23
//
//  Description:                                              
//   
//                                                                           
//  Copyright: 
//    (C) 2025 Thorsten Brach. All rights reserved                                                                                                                                            
//             Licensed under the MIT License.
//                                                                           
//  Disclaimer:                                                                           
//    This project is provided without any guarantee and can be used for   
//    private and commercial purposes. Any use is at the user’s 
//    own risk and responsibility.
//
// -------------------------------------------------------------------------
VAR_INPUT
  AxisExternalUsed : BYTE;
END_VAR

            ByteToAxisExternalUsed.E1 := AxisExternalUsed.1;
ByteToAxisExternalUsed.E2 := AxisExternalUsed.2;
ByteToAxisExternalUsed.E3 := AxisExternalUsed.3;
ByteToAxisExternalUsed.E4 := AxisExternalUsed.4;
ByteToAxisExternalUsed.E5 := AxisExternalUsed.5;
ByteToAxisExternalUsed.E6 := AxisExternalUsed.6;
          
END_FUNCTION

FUNCTION ByteToAxisJointUnit : AxisJointUnit
// ------------------------------------------------------------------------- 
//  SRCI Robot Library                                                
// ------------------------------------------------------------------------- 
//                                                                           
//  Object:      ByteToAxisJointUnit                                      
//  Author:      Thorsten Brach                                                
//  Date:        2025-03-23
//
//  Description:                                              
//   
//                                                                           
//  Copyright: 
//    (C) 2025 Thorsten Brach. All rights reserved                                                                                                                                            
//             Licensed under the MIT License.
//                                                                           
//  Disclaimer:                                                                           
//    This project is provided without any guarantee and can be used for   
//    private and commercial purposes. Any use is at the user’s 
//    own risk and responsibility.
//
// -------------------------------------------------------------------------
VAR_INPUT
  AxisJointUnit : BYTE;
END_VAR

            ByteToAxisJointUnit.J2.0 := AxisJointUnit.1;
ByteToAxisJointUnit.J2.0 := AxisJointUnit.2;
ByteToAxisJointUnit.J3.0 := AxisJointUnit.3;
ByteToAxisJointUnit.J4.0 := AxisJointUnit.4;
ByteToAxisJointUnit.J5.0 := AxisJointUnit.5;
ByteToAxisJointUnit.J6.0 := AxisJointUnit.6;
          
END_FUNCTION

FUNCTION ByteToAxisJointUsed : AxisJointUsed
// ------------------------------------------------------------------------- 
//  SRCI Robot Library                                                
// ------------------------------------------------------------------------- 
//                                                                           
//  Object:      ByteToAxisJointUsed                                       
//  Author:      Thorsten Brach                                                
//  Date:        2025-03-23
//
//  Description:                                              
//   
//                                                                           
//  Copyright: 
//    (C) 2025 Thorsten Brach. All rights reserved                                                                                                                                            
//             Licensed under the MIT License.
//                                                                           
//  Disclaimer:                                                                           
//    This project is provided without any guarantee and can be used for   
//    private and commercial purposes. Any use is at the user’s 
//    own risk and responsibility.
//
// -------------------------------------------------------------------------
VAR_INPUT
  AxisJointUsed : BYTE;
END_VAR

            ByteToAxisJointUsed.J1 := AxisJointUsed.1;
ByteToAxisJointUsed.J2 := AxisJointUsed.2;
ByteToAxisJointUsed.J3 := AxisJointUsed.3;
ByteToAxisJointUsed.J4 := AxisJointUsed.4;
ByteToAxisJointUsed.J5 := AxisJointUsed.5;
ByteToAxisJointUsed.J6 := AxisJointUsed.6;
          
END_FUNCTION

FUNCTION ByteToFragmentAction : FragmentAction
// ------------------------------------------------------------------------- 
//  SRCI Robot Library                                                
// ------------------------------------------------------------------------- 
//                                                                           
//  Object:      FragmentActionToByte                                       
//  Author:      Thorsten Brach                                                
//  Date:        2024-11-05
//
//  Description:                                              
//   
//                                                                           
//  Copyright: 
//    (C) 2024 Thorsten Brach. All rights reserved                                                                                                                                            
//             Licensed under the MIT License.
//                                                                           
//  Disclaimer:                                                                           
//    This project is provided without any guarantee and can be used for   
//    private and commercial purposes. Any use is at the user’s 
//    own risk and responsibility.
//
// -------------------------------------------------------------------------
VAR_INPUT
  FragmentAction : BYTE;
END_VAR

            ByteToFragmentAction.Complete:= FragmentAction.0; 
ByteToFragmentAction.Reset   := FragmentAction.1;   
ByteToFragmentAction.Clear   := FragmentAction.2;   
ByteToFragmentAction.BIT03   := FragmentAction.3;   
ByteToFragmentAction.BIT04   := FragmentAction.4;   
ByteToFragmentAction.BIT05   := FragmentAction.5;   
ByteToFragmentAction.BIT06   := FragmentAction.6;   
ByteToFragmentAction.BIT07   := FragmentAction.7;   
          
END_FUNCTION

FUNCTION ByteToVersion : VersionStruct
// ------------------------------------------------------------------------- 
//  SRCI Robot Library                                                
// ------------------------------------------------------------------------- 
//                                                                           
//  Object:      ByteToVersion                                       
//  Author:      Thorsten Brach                                                
//  Date:        2024-09-11
//
//  Description:                                              
//   
//                                                                           
//  Copyright: 
//    (C) 2024 Thorsten Brach. All rights reserved                                                                                                                                            
//             Licensed under the MIT License.
//                                                                           
//  Disclaimer:                                                                           
//    This project is provided without any guarantee and can be used for   
//    private and commercial purposes. Any use is at the user’s 
//    own risk and responsibility.
//
// -------------------------------------------------------------------------
VAR_INPUT
  /// Version
  Value : BYTE;
END_VAR

VAR
  _tmpByte : BYTE;
END_VAR

            // Minor version  • Features
//                • 0..31 minor versions
ByteToVersion.MinorVersion.0 := Value.0;
ByteToVersion.MinorVersion.1 := Value.1;
ByteToVersion.MinorVersion.2 := Value.2;
ByteToVersion.MinorVersion.3 := Value.3;
ByteToVersion.MinorVersion.4 := Value.4;

// Major version  • Breaking change
//                • 0..7 major versions
ByteToVersion.MajorVersion.0 := Value.5;
ByteToVersion.MajorVersion.1 := Value.6;
ByteToVersion.MajorVersion.2 := Value.7;
          
END_FUNCTION

FUNCTION CombineBytesToUint : UINT
// ------------------------------------------------------------------------- 
//  SRCI Robot Library                                                
// ------------------------------------------------------------------------- 
//                                                                           
//  Object:      CombineBytes                                       
//  Author:      Thorsten Brach                                                
//  Date:        2024-09-03
//
//  Description:                                              
//   
//                                                                           
//  Copyright: 
//    (C) 2024 Thorsten Brach. All rights reserved                                                                                                                                            
//             Licensed under the MIT License.
//                                                                           
//  Disclaimer:                                                                           
//    This project is provided without any guarantee and can be used for   
//    private and commercial purposes. Any use is at the user’s 
//    own risk and responsibility.
//
// -------------------------------------------------------------------------
VAR_INPUT
  /// Byte to add as high byte
  HiByte : BYTE;
  /// Byte to add as low byte
  LoByte : BYTE;
END_VAR

            CombineBytesToUint.0  := LoByte.0;
CombineBytesToUint.1  := LoByte.1;
CombineBytesToUint.2  := LoByte.2;
CombineBytesToUint.3  := LoByte.3;
CombineBytesToUint.4  := LoByte.4;
CombineBytesToUint.5  := LoByte.5;
CombineBytesToUint.6  := LoByte.6;
CombineBytesToUint.7  := LoByte.7;

CombineBytesToUint.8  := HiByte.0;
CombineBytesToUint.9  := HiByte.1;
CombineBytesToUint.10 := HiByte.2;
CombineBytesToUint.11 := HiByte.3;
CombineBytesToUint.12 := HiByte.4;
CombineBytesToUint.13 := HiByte.5;
CombineBytesToUint.14 := HiByte.6;
CombineBytesToUint.15 := HiByte.7;
          
END_FUNCTION

FUNCTION CombineHalfBytes : USINT
// ------------------------------------------------------------------------- 
//  SRCI Robot Library                                                
// ------------------------------------------------------------------------- 
//                                                                           
//  Object:      CombineHalfBytes                                       
//  Author:      Thorsten Brach                                                
//  Date:        2024-06-01
//
//  Description:                                              
//   
//                                                                           
//  Copyright: 
//    (C) 2024 Thorsten Brach. All rights reserved                                                                                                                                            
//             Licensed under the MIT License.
//                                                                           
//  Disclaimer:                                                                           
//    This project is provided without any guarantee and can be used for   
//    private and commercial purposes. Any use is at the user’s 
//    own risk and responsibility.
//
// -------------------------------------------------------------------------
VAR_INPUT
  /// Half-Byte to add to the upper 4 Bit
  HalfByteHi : BYTE;
  /// Half-Byte to add to the lower 4 Bit
  HalfByteLo : BYTE;
END_VAR

            // merage ParSeq and Priority to combined variable
CombineHalfBytes.0 := HalfByteLo.0;
CombineHalfBytes.1 := HalfByteLo.1;
CombineHalfBytes.2 := HalfByteLo.2;
CombineHalfBytes.3 := HalfByteLo.3;

CombineHalfBytes.4 := HalfByteHi.0;
CombineHalfBytes.5 := HalfByteHi.1;
CombineHalfBytes.6 := HalfByteHi.2;
CombineHalfBytes.7 := HalfByteHi.3;
          
END_FUNCTION

FUNCTION CombineHalfSints : USINT
// ------------------------------------------------------------------------- 
//  SRCI Robot Library                                                
// ------------------------------------------------------------------------- 
//                                                                           
//  Object:      CombineHalfSints                                       
//  Author:      Thorsten Brach                                                
//  Date:        2025-02-02
//
//  Description:                                              
//   
//                                                                           
//  Copyright: 
//    (C) 2025 Thorsten Brach. All rights reserved                                                                                                                                            
//             Licensed under the MIT License.
//                                                                           
//  Disclaimer:                                                                           
//    This project is provided without any guarantee and can be used for   
//    private and commercial purposes. Any use is at the user’s 
//    own risk and responsibility.
//
// -------------------------------------------------------------------------
VAR_INPUT
  /// Half-Sint to add to the upper 4 Bit
  HalfSintHi : SINT;
  /// Half-Sint to add to the lower 4 Bit
  HalfSintLo : SINT;
END_VAR

            // merage ParSeq and Priority to combined variable
CombineHalfSints.0 := HalfSintLo.0;
CombineHalfSints.1 := HalfSintLo.1;
CombineHalfSints.2 := HalfSintLo.2;
CombineHalfSints.3 := HalfSintLo.3;

CombineHalfSints.4 := HalfSintHi.0;
CombineHalfSints.5 := HalfSintHi.1;
CombineHalfSints.6 := HalfSintHi.2;
CombineHalfSints.7 := HalfSintHi.3;
          
END_FUNCTION

FUNCTION DwordToRaStatusWord : RaStatusWord
// ------------------------------------------------------------------------- 
//  SRCI Robot Library                                                
// ------------------------------------------------------------------------- 
//                                                                           
//  Object:      DwordToRaStatusWord                                       
//  Author:      Thorsten Brach                                                
//  Date:        2024-11-16
//
//  Description:                                              
//   
//                                                                           
//  Copyright: 
//    (C) 2024 Thorsten Brach. All rights reserved                                                                                                                                            
//             Licensed under the MIT License.
//                                                                           
//  Disclaimer:                                                                           
//    This project is provided without any guarantee and can be used for   
//    private and commercial purposes. Any use is at the user’s 
//    own risk and responsibility.
//
// -------------------------------------------------------------------------
VAR_INPUT
  /// Value
  Value : DWORD;
END_VAR

            DwordToRaStatusWord.IsMoving                 := Value.00;
DwordToRaStatusWord.PrimarySequencePaused    := Value.01;
DwordToRaStatusWord.InPrimaryPos             := Value.02;
DwordToRaStatusWord.SecondarySequenceActive  := Value.03;
DwordToRaStatusWord.IsBlending               := Value.04;
DwordToRaStatusWord.ErrorPending             := Value.05;
DwordToRaStatusWord.RestartInProgress        := Value.06;
DwordToRaStatusWord.Enabled                  := Value.07;
DwordToRaStatusWord.RaSequenceState.0        := Value.08;
DwordToRaStatusWord.RaSequenceState.1        := Value.09;
DwordToRaStatusWord.OperationMode.0          := Value.10;
DwordToRaStatusWord.OperationMode.1          := Value.11;
DwordToRaStatusWord.OperationMode.2          := Value.12;
DwordToRaStatusWord.CollisionDetectedEnabled := Value.13;
DwordToRaStatusWord.CollisionDetected        := Value.14;
DwordToRaStatusWord.RestartRequested         := Value.15;
DwordToRaStatusWord.Accelerating             := Value.16;
DwordToRaStatusWord.Decelerating             := Value.17;
DwordToRaStatusWord.ConstantVelocity         := Value.18;
DwordToRaStatusWord.Bit19                    := Value.19;
DwordToRaStatusWord.Bit20                    := Value.20;
DwordToRaStatusWord.Bit21                    := Value.21;
DwordToRaStatusWord.Bit22                    := Value.22;
DwordToRaStatusWord.Bit23                    := Value.23;
DwordToRaStatusWord.Bit24                    := Value.24;
DwordToRaStatusWord.Bit25                    := Value.25;
DwordToRaStatusWord.Bit26                    := Value.26;
DwordToRaStatusWord.Bit27                    := Value.27;
DwordToRaStatusWord.Bit28                    := Value.28;
DwordToRaStatusWord.Bit29                    := Value.29;
DwordToRaStatusWord.Bit30                    := Value.30;
DwordToRaStatusWord.Bit31                    := Value.31;
          
END_FUNCTION

FUNCTION FragmentActionToByte : BYTE
// ------------------------------------------------------------------------- 
//  SRCI Robot Library                                                
// ------------------------------------------------------------------------- 
//                                                                           
//  Object:      FragmentActionToByte                                       
//  Author:      Thorsten Brach                                                
//  Date:        2024-06-01
//
//  Description:                                              
//   
//                                                                           
//  Copyright: 
//    (C) 2024 Thorsten Brach. All rights reserved                                                                                                                                            
//             Licensed under the MIT License.
//                                                                           
//  Disclaimer:                                                                           
//    This project is provided without any guarantee and can be used for   
//    private and commercial purposes. Any use is at the user’s 
//    own risk and responsibility.
//
// -------------------------------------------------------------------------
VAR_INPUT
  FragmentAction : FragmentAction;
END_VAR

            FragmentActionToByte.0 := FragmentAction.Complete;
FragmentActionToByte.1 := FragmentAction.Reset;
FragmentActionToByte.2 := FragmentAction.Clear;
FragmentActionToByte.3 := FragmentAction.BIT03;
FragmentActionToByte.4 := FragmentAction.BIT04;
FragmentActionToByte.5 := FragmentAction.BIT05;
FragmentActionToByte.6 := FragmentAction.BIT06;
FragmentActionToByte.7 := FragmentAction.BIT07;
          
END_FUNCTION

FUNCTION PERCENT_INT_TO_REAL : REAL
// ------------------------------------------------------------------------- 
//  SRCI Robot Library                                                
// ------------------------------------------------------------------------- 
//                                                                           
//  Object:      PERCENT_INT_TO_REAL                                       
//  Author:      Thorsten Brach                                                
//  Date:        2025-02-07
//
//  Description:                                              
//   
//                                                                           
//  Copyright: 
//    (C) 2025 Thorsten Brach. All rights reserved                                                                                                                                            
//             Licensed under the MIT License.
//                                                                           
//  Disclaimer:                                                                           
//    This project is provided without any guarantee and can be used for   
//    private and commercial purposes. Any use is at the user’s 
//    own risk and responsibility.
//
// -------------------------------------------------------------------------
VAR_INPUT
  /// Percent value to convert 
  Value    : INT;
  /// value is an optional parameter ?  
  IsOptional : BOOL;
END_VAR

            IF (( Value = 16#FFFF_FFFF ) AND (IsOptional)) OR // 16#FFFF_FFFF for not supported values
   (( Value = 16#0000_FFFF ) AND (IsOptional))    // 16#0000_FFFF for not supported values 
THEN
  PERCENT_INT_TO_REAL := -1.0;
ELSE
  PERCENT_INT_TO_REAL := INT_TO_REAL(Value) / RobotLibraryConstants.REAL_CONVERSION_FACTOR;   
END_IF
          
END_FUNCTION

FUNCTION PERCENT_UINT_TO_REAL : REAL
// ------------------------------------------------------------------------- 
//  SRCI Robot Library                                                
// ------------------------------------------------------------------------- 
//                                                                           
//  Object:      PERCENT_UINT_TO_REAL                                       
//  Author:      Thorsten Brach                                                
//  Date:        2025-04-02
//
//  Description:                                              
//   
//                                                                           
//  Copyright: 
//    (C) 2025 Thorsten Brach. All rights reserved                                                                                                                                            
//             Licensed under the MIT License.
//                                                                           
//  Disclaimer:                                                                           
//    This project is provided without any guarantee and can be used for   
//    private and commercial purposes. Any use is at the user’s 
//    own risk and responsibility.
//
// -------------------------------------------------------------------------
VAR_INPUT
  /// Percent value to convert 
  Value    : UINT;
  /// value is an optional parameter ?  
  IsOptional : BOOL;
END_VAR

            IF (( Value = 16#FFFF_FFFF ) AND (IsOptional)) OR // 16#FFFF_FFFF for not supported values
   (( Value = 16#0000_FFFF ) AND (IsOptional))    // 16#0000_FFFF for not supported values 
THEN
  PERCENT_UINT_TO_REAL := -1.0;
  RETURN;
END_IF

PERCENT_UINT_TO_REAL := UINT_TO_REAL(Value) / RobotLibraryConstants.REAL_CONVERSION_FACTOR; 
          
END_FUNCTION

FUNCTION PlcOptionalCyclicToUint : UINT
// ------------------------------------------------------------------------- 
//  SRCI Robot Library                                                
// ------------------------------------------------------------------------- 
//                                                                           
//  Object:      PlcOptionalCyclicToUint                                       
//  Author:      Thorsten Brach                                                
//  Date:        2024-11-30
//
//  Description:                                              
//   
//                                                                           
//  Copyright: 
//    (C) 2024 Thorsten Brach. All rights reserved                                                                                                                                            
//             Licensed under the MIT License.
//                                                                           
//  Disclaimer:                                                                           
//    This project is provided without any guarantee and can be used for   
//    private and commercial purposes. Any use is at the user’s 
//    own risk and responsibility.
//
// -------------------------------------------------------------------------
VAR_INPUT
  OptionalCyclic : AxesGroupParameterPlcOptionalCyclic;
END_VAR

            PlcOptionalCyclicToUint.00 := OptionalCyclic.UseCallSubprogram;
PlcOptionalCyclicToUint.01 := OptionalCyclic.UseCartesianPosition;
PlcOptionalCyclicToUint.02 := OptionalCyclic.UseJointPosition;
PlcOptionalCyclicToUint.03 := OptionalCyclic.UseForce;
PlcOptionalCyclicToUint.04 := OptionalCyclic.Bit04;
PlcOptionalCyclicToUint.05 := OptionalCyclic.Bit05;
PlcOptionalCyclicToUint.06 := OptionalCyclic.Bit06;
PlcOptionalCyclicToUint.07 := OptionalCyclic.Bit07;  
PlcOptionalCyclicToUint.08 := OptionalCyclic.UseTwoSequences;
PlcOptionalCyclicToUint.09 := OptionalCyclic.UseCartesianPositionExt;
PlcOptionalCyclicToUint.10 := OptionalCyclic.UseJointPositionExt;
PlcOptionalCyclicToUint.11 := OptionalCyclic.Bit11;
PlcOptionalCyclicToUint.12 := OptionalCyclic.Bit12;
PlcOptionalCyclicToUint.13 := OptionalCyclic.Bit13;
PlcOptionalCyclicToUint.14 := OptionalCyclic.Bit14;
PlcOptionalCyclicToUint.15 := OptionalCyclic.Bit15;  

          
END_FUNCTION

FUNCTION REAL_TO_PERCENT_INT : INT
// ------------------------------------------------------------------------- 
//  SRCI Robot Library                                                
// ------------------------------------------------------------------------- 
//                                                                           
//  Object:      REAL_TO_PERCENT_INT                                       
//  Author:      Thorsten Brach                                                
//  Date:        2025-02-07
//
//  Description:                                              
//   
//                                                                           
//  Copyright: 
//    (C) 2025 Thorsten Brach. All rights reserved                                                                                                                                            
//             Licensed under the MIT License.
//                                                                           
//  Disclaimer:                                                                           
//    This project is provided without any guarantee and can be used for   
//    private and commercial purposes. Any use is at the user’s 
//    own risk and responsibility.
//
// -------------------------------------------------------------------------
VAR_INPUT
  /// Percent value to convert 
  Value      : REAL;
  /// value is an optional parameter ?  
  IsOptional : BOOL;
END_VAR

            IF ( Value = -1.0)  AND (IsOptional)// 16#FFFF for not supported values 
THEN
  REAL_TO_PERCENT_INT := UINT_TO_INT(16#FFFF);
  RETURN;
END_IF

REAL_TO_PERCENT_INT := REAL_TO_INT(Value * RobotLibraryConstants.REAL_CONVERSION_FACTOR);
          
END_FUNCTION

FUNCTION REAL_TO_PERCENT_UINT : UINT
// ------------------------------------------------------------------------- 
//  SRCI Robot Library                                                
// ------------------------------------------------------------------------- 
//                                                                           
//  Object:      REAL_TO_PERCENT_UINT                                       
//  Author:      Thorsten Brach                                                
//  Date:        2025-02-07
//
//  Description:                                              
//   
//                                                                           
//  Copyright: 
//    (C) 2025 Thorsten Brach. All rights reserved                                                                                                                                            
//             Licensed under the MIT License.
//                                                                           
//  Disclaimer:                                                                           
//    This project is provided without any guarantee and can be used for   
//    private and commercial purposes. Any use is at the user’s 
//    own risk and responsibility.
//
// -------------------------------------------------------------------------
VAR_INPUT
  /// Percent value to convert 
  Value      : REAL;
  /// value is an optional parameter ?  
  IsOptional : BOOL;
END_VAR

            IF ( Value = -1.0)  AND (IsOptional)// 16#FFFF for not supported values 
THEN
  REAL_TO_PERCENT_UINT := 16#FFFF;
  RETURN;
END_IF

REAL_TO_PERCENT_UINT := REAL_TO_UINT(Value * RobotLibraryConstants.REAL_CONVERSION_FACTOR);
          
END_FUNCTION

FUNCTION RobOptionalCyclicToUint : UINT
// ------------------------------------------------------------------------- 
//  SRCI Robot Library                                                
// ------------------------------------------------------------------------- 
//                                                                           
//  Object:      RobOptionalCyclicToUint                                       
//  Author:      Thorsten Brach                                                
//  Date:        2024-11-30
//
//  Description:                                              
//   
//                                                                           
//  Copyright: 
//    (C) 2024 Thorsten Brach. All rights reserved                                                                                                                                            
//             Licensed under the MIT License.
//                                                                           
//  Disclaimer:                                                                           
//    This project is provided without any guarantee and can be used for   
//    private and commercial purposes. Any use is at the user’s 
//    own risk and responsibility.
//
// -------------------------------------------------------------------------
VAR_INPUT
  OptionalCyclic : AxesGroupParameterRobOptionalCyclic;
END_VAR

            RobOptionalCyclicToUint.00 := OptionalCyclic.UseCallSubprogram;      
RobOptionalCyclicToUint.01 := OptionalCyclic.UseCartesianPosition;   
RobOptionalCyclicToUint.02 := OptionalCyclic.UseJointPosition;       
RobOptionalCyclicToUint.03 := OptionalCyclic.UseForce;               
RobOptionalCyclicToUint.04 := OptionalCyclic.UseCurrent;             
RobOptionalCyclicToUint.05 := OptionalCyclic.Bit05;                  
RobOptionalCyclicToUint.06 := OptionalCyclic.Bit06;                  
RobOptionalCyclicToUint.07 := OptionalCyclic.Bit07;                  
RobOptionalCyclicToUint.08 := OptionalCyclic.UseTwoSequences;        
RobOptionalCyclicToUint.09 := OptionalCyclic.UseCartesianPositionExt;
RobOptionalCyclicToUint.10 := OptionalCyclic.UseJointPositionExt;    
RobOptionalCyclicToUint.11 := OptionalCyclic.UseForceExt;            
RobOptionalCyclicToUint.12 := OptionalCyclic.UseCurrentExt;          
RobOptionalCyclicToUint.13 := OptionalCyclic.Bit13;                  
RobOptionalCyclicToUint.14 := OptionalCyclic.Bit14;                  
RobOptionalCyclicToUint.15 := OptionalCyclic.Bit15;                  

          
END_FUNCTION

FUNCTION SyncModesToDataEnableSync : DataEnableSync
// ------------------------------------------------------------------------- 
//  SRCI Robot Library                                                
// ------------------------------------------------------------------------- 
//                                                                           
//  Object:      SyncModesToDataEnableSync                                       
//  Author:      Thorsten Brach                                                
//  Date:        2025-04-22
//
//  Description:                                              
//   
//                                                                           
//  Copyright: 
//    (C) 2025 Thorsten Brach. All rights reserved                                                                                                                                            
//             Licensed under the MIT License.
//                                                                           
//  Disclaimer:                                                                           
//    This project is provided without any guarantee and can be used for   
//    private and commercial purposes. Any use is at the user’s 
//    own risk and responsibility.
//
// -------------------------------------------------------------------------
VAR_INPUT
  /// Synchronization Modes
  Value : SynchronizationModes;  
END_VAR

            SyncModesToDataEnableSync.EnableSyncTool              := Value.Tool             [SyncTime.DURING_START_UP] > SyncMode.NO_SYNCHRONIZATION OR
                                                         Value.Tool             [SyncTime. AFTER_START_UP] > SyncMode.NO_SYNCHRONIZATION;                                                  
SyncModesToDataEnableSync.EnableSyncFrame             := Value.Frame            [SyncTime.DURING_START_UP] > SyncMode.NO_SYNCHRONIZATION OR
                                                         Value.Frame            [SyncTime. AFTER_START_UP] > SyncMode.NO_SYNCHRONIZATION;
SyncModesToDataEnableSync.EnableSyncLoad              := Value.Load             [SyncTime.DURING_START_UP] > SyncMode.NO_SYNCHRONIZATION OR
                                                         Value.Load             [SyncTime. AFTER_START_UP] > SyncMode.NO_SYNCHRONIZATION;
SyncModesToDataEnableSync.EnableSyncWorkArea          := Value.WorkAreas        [SyncTime.DURING_START_UP] > SyncMode.NO_SYNCHRONIZATION OR
                                                         Value.WorkAreas        [SyncTime. AFTER_START_UP] > SyncMode.NO_SYNCHRONIZATION;
SyncModesToDataEnableSync.EnableSyncSWLimits          := Value.SWLimits         [SyncTime.DURING_START_UP] > SyncMode.NO_SYNCHRONIZATION OR
                                                         Value.SWLimits         [SyncTime. AFTER_START_UP] > SyncMode.NO_SYNCHRONIZATION;
SyncModesToDataEnableSync.EnableSyncDefaultDynamics   := Value.DefaultDynamics  [SyncTime.DURING_START_UP] > SyncMode.NO_SYNCHRONIZATION OR
                                                         Value.DefaultDynamics  [SyncTime. AFTER_START_UP] > SyncMode.NO_SYNCHRONIZATION;                                        
SyncModesToDataEnableSync.EnableSyncReferenceDynamics := Value.ReferenceDynamics[SyncTime.DURING_START_UP] > SyncMode.NO_SYNCHRONIZATION OR
                                                         Value.ReferenceDynamics[SyncTime. AFTER_START_UP] > SyncMode.NO_SYNCHRONIZATION;
          
END_FUNCTION

FUNCTION VersionToByte : BYTE
// ------------------------------------------------------------------------- 
//  SRCI Robot Library                                                
// ------------------------------------------------------------------------- 
//                                                                           
//  Object:      VersionToByte                                       
//  Author:      Thorsten Brach                                                
//  Date:        2024-06-01
//
//  Description:                                              
//   
//                                                                           
//  Copyright: 
//    (C) 2024 Thorsten Brach. All rights reserved                                                                                                                                            
//             Licensed under the MIT License.
//                                                                           
//  Disclaimer:                                                                           
//    This project is provided without any guarantee and can be used for   
//    private and commercial purposes. Any use is at the user’s 
//    own risk and responsibility.
//
// -------------------------------------------------------------------------
VAR_INPUT
  /// Version
  Value : VersionStruct;
END_VAR

VAR
  _tmpByte : BYTE;
END_VAR

            // Minor version  • Features
//                • 0..31 minor versions
VersionToByte.0 := Value.MinorVersion.0;
VersionToByte.1 := Value.MinorVersion.1;
VersionToByte.2 := Value.MinorVersion.2;
VersionToByte.3 := Value.MinorVersion.3;
VersionToByte.4 := Value.MinorVersion.4;

// Major version  • Breaking change
//                • 0..7 major versions
VersionToByte.5 := Value.MajorVersion.0;
VersionToByte.6 := Value.MajorVersion.1;
VersionToByte.7 := Value.MajorVersion.2;
          
END_FUNCTION

FUNCTION WordToArmConfigElbow : ArmConfigElbow
// ------------------------------------------------------------------------- 
//  SRCI Robot Library                                                
// ------------------------------------------------------------------------- 
//                                                                           
//  Object:      WordToArmConfigElbow                                       
//  Author:      Thorsten Brach                                                
//  Date:        2024-12-24
//
//  Description:                                              
//   
//                                                                           
//  Copyright: 
//    (C) 2024 Thorsten Brach. All rights reserved                                                                                                                                            
//             Licensed under the MIT License.
//                                                                           
//  Disclaimer:                                                                           
//    This project is provided without any guarantee and can be used for   
//    private and commercial purposes. Any use is at the user’s 
//    own risk and responsibility.
//
// -------------------------------------------------------------------------
VAR_INPUT
  /// Value
  Value : WORD;
END_VAR

VAR
  _tmpByte : BYTE;
END_VAR

            IF ( RobotLibraryParameter.SWAP_BYTE_ORDER)
THEN
  Value := SwapWord(Value);
END_IF

IF (Value.1)
THEN
  WordToArmConfigElbow := ArmConfigElbow.DOWN;
ELSE
  WordToArmConfigElbow := ArmConfigElbow.UP;  
END_IF


          
END_FUNCTION

FUNCTION WordToArmConfigShoulder : ArmConfigShoulder
// ------------------------------------------------------------------------- 
//  SRCI Robot Library                                                
// ------------------------------------------------------------------------- 
//                                                                           
//  Object:      WordToArmConfigShoulder                                       
//  Author:      Thorsten Brach                                                
//  Date:        2024-12-24
//
//  Description:                                              
//   
//                                                                           
//  Copyright: 
//    (C) 2024 Thorsten Brach. All rights reserved                                                                                                                                            
//             Licensed under the MIT License.
//                                                                           
//  Disclaimer:                                                                           
//    This project is provided without any guarantee and can be used for   
//    private and commercial purposes. Any use is at the user’s 
//    own risk and responsibility.
//
// -------------------------------------------------------------------------
VAR_INPUT
  /// Value
  Value : WORD;
END_VAR

VAR
  _tmpByte : BYTE;
END_VAR

            IF ( RobotLibraryParameter.SWAP_BYTE_ORDER)
THEN
  Value := SwapWord(Value);
END_IF

IF (Value.0)
THEN
  WordToArmConfigShoulder := ArmConfigShoulder.BACK;
ELSE
  WordToArmConfigShoulder := ArmConfigShoulder.FRONT;  
END_IF


          
END_FUNCTION

FUNCTION WordToArmConfigWrist : ArmConfigWrist
// ------------------------------------------------------------------------- 
//  SRCI Robot Library                                                
// ------------------------------------------------------------------------- 
//                                                                           
//  Object:      WordToArmConfigWrist                                       
//  Author:      Thorsten Brach                                                
//  Date:        2024-12-24
//
//  Description:                                              
//   
//                                                                           
//  Copyright: 
//    (C) 2024 Thorsten Brach. All rights reserved                                                                                                                                            
//             Licensed under the MIT License.
//                                                                           
//  Disclaimer:                                                                           
//    This project is provided without any guarantee and can be used for   
//    private and commercial purposes. Any use is at the user’s 
//    own risk and responsibility.
//
// -------------------------------------------------------------------------
VAR_INPUT
  /// Value
  Value : WORD;
END_VAR

VAR
  _tmpByte : BYTE;
END_VAR

            IF ( RobotLibraryParameter.SWAP_BYTE_ORDER)
THEN
  Value := SwapWord(Value);
END_IF

IF (Value.2)
THEN
  WordToArmConfigWrist := ArmConfigWrist.FLIP;
ELSE
  WordToArmConfigWrist := ArmConfigWrist.NON_FLIP;  
END_IF


          
END_FUNCTION

FUNCTION ABORTING_MODE_TO_STRING : STRING
// ------------------------------------------------------------------------- 
//  SRCI Robot Library                                                
// ------------------------------------------------------------------------- 
//                                                                           
//  Object:      ABORTING_MODE_TO_STRING                                       
//  Author:      Thorsten Brach                                                
//  Date:        2025-02-23
//
//  Description:                                              
//   
//                                                                           
//  Copyright: 
//    (C) 2025 Thorsten Brach. All rights reserved                                                                                                                                            
//             Licensed under the MIT License.
//                                                                           
//  Disclaimer:                                                                           
//    This project is provided without any guarantee and can be used for   
//    private and commercial purposes. Any use is at the user’s 
//    own risk and responsibility.
//
// -------------------------------------------------------------------------
VAR_INPUT
  /// AbortingMode
  Value : AbortingMode;
END_VAR

            CASE Value 
OF
  AbortingMode.BUFFER : ABORTING_MODE_TO_STRING := StrReplace('BUFFER ({0})','{0}' , SINT_TO_STRING(Value));
  AbortingMode.ABORT  : ABORTING_MODE_TO_STRING := StrReplace('ABORT ({0})' ,'{0}' , SINT_TO_STRING(Value));
ELSE
  ABORTING_MODE_TO_STRING := CONCAT('ABORTING_MODE_TO_STRING Function: Error -> no parsing for value ', SINT_TO_STRING(Value));
END_CASE
          
END_FUNCTION

FUNCTION ALARM_MESSAGE_TO_STRING : STRING(RobotLibraryParameter.MESSAGE_TEXT_LEN)
// ------------------------------------------------------------------------- 
//  SRCI Robot Library                                                
// ------------------------------------------------------------------------- 
//                                                                           
//  Object:      ALARM_MESSAGE_TO_STRING                                       
//  Author:      Thorsten Brach                                                
//  Date:        2025-03-31
//
//  Description:                                              
//   
//                                                                           
//  Copyright: 
//    (C) 2025 Thorsten Brach. All rights reserved                                                                                                                                            
//             Licensed under the MIT License.
//                                                                           
//  Disclaimer:                                                                           
//    This project is provided without any guarantee and can be used for   
//    private and commercial purposes. Any use is at the user’s 
//    own risk and responsibility.
//
// -------------------------------------------------------------------------
VAR_INPUT
  /// AlarmMessag
  Message : AlarmMessage;
END_VAR
VAR CONSTANT
  /// Carrage return and line feed
  CRLF       : STRING := '$R$N';
END_VAR

            ALARM_MESSAGE_TO_STRING := CONCAT    (ALARM_MESSAGE_TO_STRING, DATE_TO_STRING(Message.Timestamp.SystemDate));
ALARM_MESSAGE_TO_STRING := CONCAT    (ALARM_MESSAGE_TO_STRING, '-');
ALARM_MESSAGE_TO_STRING := CONCAT    (ALARM_MESSAGE_TO_STRING, TOD_TO_STRING (Message.Timestamp.SystemTime));
ALARM_MESSAGE_TO_STRING := StrReplace(ALARM_MESSAGE_TO_STRING, 'TOD#','' );
ALARM_MESSAGE_TO_STRING := StrReplace(ALARM_MESSAGE_TO_STRING, 'D#', '' );
ALARM_MESSAGE_TO_STRING := CONCAT    (ALARM_MESSAGE_TO_STRING, ':');
ALARM_MESSAGE_TO_STRING := CONCAT    (ALARM_MESSAGE_TO_STRING, MESSAGE_TYPE_TO_STRING(Value := Message.MessageType, AlignString := TRUE));
ALARM_MESSAGE_TO_STRING := CONCAT    (ALARM_MESSAGE_TO_STRING, ':');
ALARM_MESSAGE_TO_STRING := CONCAT    (ALARM_MESSAGE_TO_STRING, SEVERITY_TO_STRING    ( Value := Message.Severity  , AlignString := TRUE));
ALARM_MESSAGE_TO_STRING := CONCAT    (ALARM_MESSAGE_TO_STRING, ':');
ALARM_MESSAGE_TO_STRING := CONCAT    (ALARM_MESSAGE_TO_STRING, DWORD_TO_STRING(Message.MessageCode));
ALARM_MESSAGE_TO_STRING := CONCAT    (ALARM_MESSAGE_TO_STRING, ':');
ALARM_MESSAGE_TO_STRING := CONCAT    (ALARM_MESSAGE_TO_STRING, Message.MessageText);
ALARM_MESSAGE_TO_STRING := CONCAT    (ALARM_MESSAGE_TO_STRING, CRLF);
          
END_FUNCTION

